TYPE ST_TrayMotionConfig :
STRUCT
    stX : ST_VelocityConfig;
    stZ : ST_VelocityConfig;
END_STRUCT
END_TYPE

(* stored: Version 1.1.0.1, ProductVersion 3.1.4026.20
   DUT ST_TrayMotionConfig: Id {5aabdcc9-2a58-4c5a-8639-466cba1440e8} *)
